// Writes out part of an array of bytes.
FUNCTION F_WriteRawByte : HRESULT
VAR_IN_OUT
    stCtx   : ST_WriteContext;
END_VAR
VAR_INPUT CONSTANT
    nValue  : BYTE;
END_VAR

VAR CONSTANT
    cLength : UDINT := SIZEOF(nValue);
END_VAR
VAR
    pByte   : POINTER TO BYTE;
END_VAR


F_WriteRawByte := S_OK;

IF cLength > stCtx.stState.nBufferSize - stCtx.stState.nBufferPos THEN
    F_WriteRawByte := stCtx.stState.eWriterErrorCode := E_WriterErrorCode.TruncatedMessage;
    stCtx.stState.bError := TRUE;
    RETURN;
END_IF

pByte := stCtx.stBuffer.pBuffer + stCtx.stState.nBufferPos;
pByte^ := nValue;
stCtx.stState.nBufferPos := stCtx.stState.nBufferPos + cLength;

END_FUNCTION

(* stored: Version 1.1.0.1
   POU F_WriteRawByte: Id {b076660d-c3ec-4678-82dc-e1aecd7132d4}, SpecialFunc None *)
